(* PLC project sfc_multi_actionblock, TiZi TiZi 1 *)

PROGRAM main
  VAR
    A : BOOL;
    B : BOOL;
  END_VAR

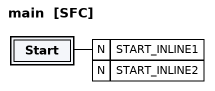
INITIAL_STEP Start:
  START_INLINE1(N);
  START_INLINE2(N);
END_STEP
ACTION START_INLINE1:
  A := TRUE;
END_ACTION
ACTION START_INLINE2:
  B := TRUE;
END_ACTION
END_PROGRAM
